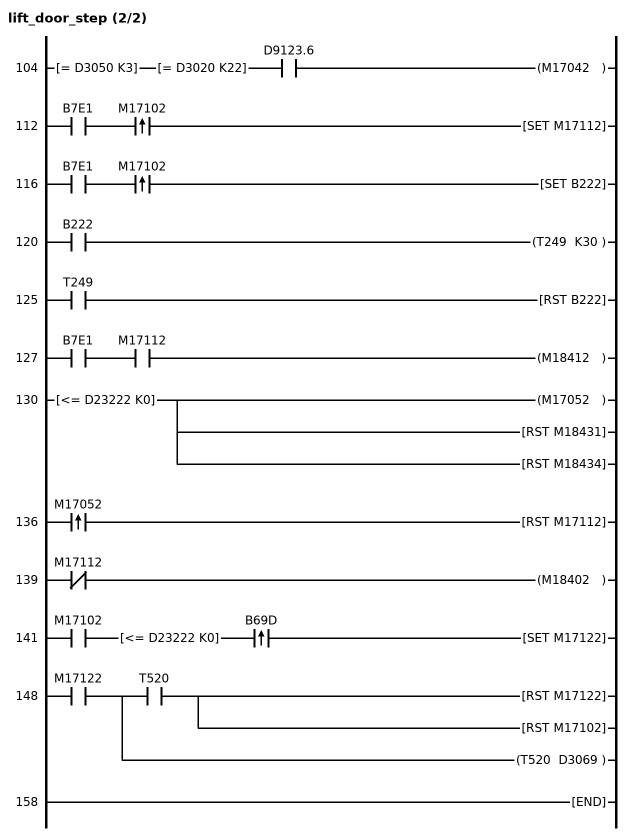
[picture p240: ladder of lift_door_step, rungs at steps 104 to 158]
104   LD=     D3050 K3
      AND=    D3020 K22
      AND     D9123.6
      OUT     M17042
112   LD      B7E1
      ANDP    M17102
      SET     M17112
116   LD      B7E1
      ANDP    M17102
      SET     B222
120   LD      B222
      OUT     T249 K30
125   LD      T249
      RST     B222
127   LD      B7E1
      AND     M17112
      OUT     M18412
130   LD<=    D23222 K0
      OUT     M17052
      RST     M18431
      RST     M18434
136   LDP     M17052
      RST     M17112
139   LDI     M17112
      OUT     M18402
141   LD      M17102
      AND<=   D23222 K0
      ANDP    B69D
      SET     M17122
148   LD      M17122
      MPS
      AND     T520
      RST     M17122
      RST     M17102
      MPP
      OUT     T520 D3069
158   END
END_PROGRAM

PROGRAM next_cap_step
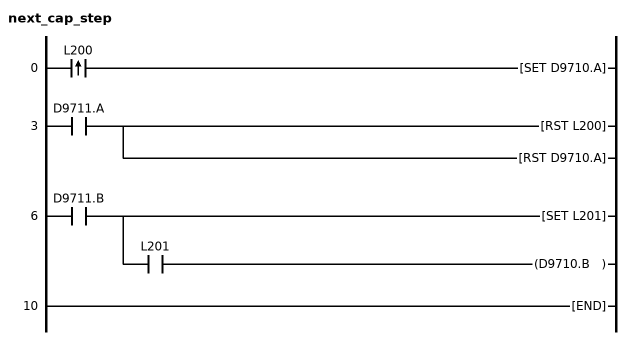
0     LDP     L200
      SET     D9710.A
3     LD      D9711.A
      RST     L200
      RST     D9710.A
6     LD      D9711.B
      SET     L201
      AND     L201
      OUT     D9710.B
10    END
END_PROGRAM

PROGRAM output
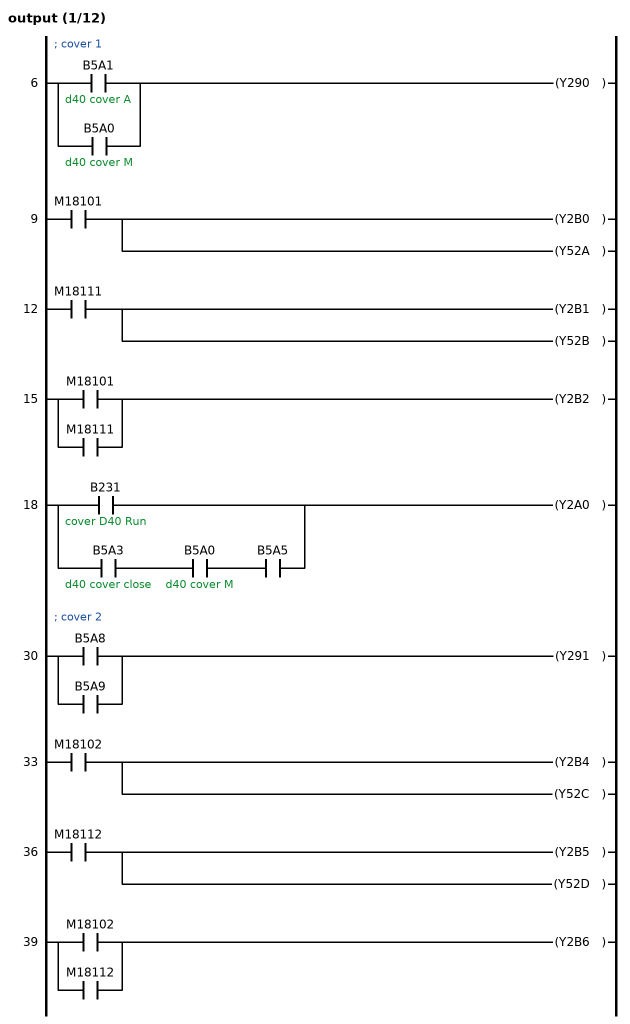
; cover 1
6     LD      B5A1  ; d40 cover A
      OR      B5A0  ; d40 cover M
      OUT     Y290
9     LD      M18101
      OUT     Y2B0
      OUT     Y52A
12    LD      M18111
      OUT     Y2B1
      OUT     Y52B
15    LD      M18101
      OR      M18111
      OUT     Y2B2
18    LD      B231  ; cover D40 Run
      LD      B5A3  ; d40 cover close
      AND     B5A0  ; d40 cover M
      AND     B5A5
      ORB
      OUT     Y2A0
; cover 2
30    LD      B5A8
      OR      B5A9
      OUT     Y291
33    LD      M18102
      OUT     Y2B4
      OUT     Y52C
36    LD      M18112
      OUT     Y2B5
      OUT     Y52D
39    LD      M18102
      OR      M18112
      OUT     Y2B6
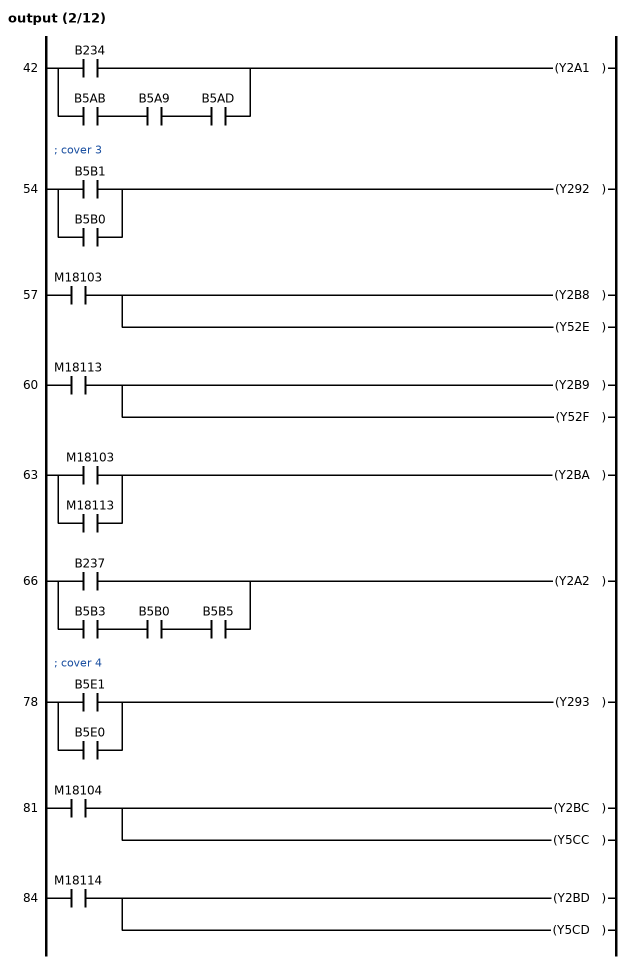
42    LD      B234
      LD      B5AB
      AND     B5A9
      AND     B5AD
      ORB
      OUT     Y2A1
; cover 3
54    LD      B5B1
      OR      B5B0
      OUT     Y292
57    LD      M18103
      OUT     Y2B8
      OUT     Y52E
60    LD      M18113
      OUT     Y2B9
      OUT     Y52F
63    LD      M18103
      OR      M18113
      OUT     Y2BA
66    LD      B237
      LD      B5B3
      AND     B5B0
      AND     B5B5
      ORB
      OUT     Y2A2
; cover 4
78    LD      B5E1
      OR      B5E0
      OUT     Y293
81    LD      M18104
      OUT     Y2BC
      OUT     Y5CC
84    LD      M18114
      OUT     Y2BD
      OUT     Y5CD
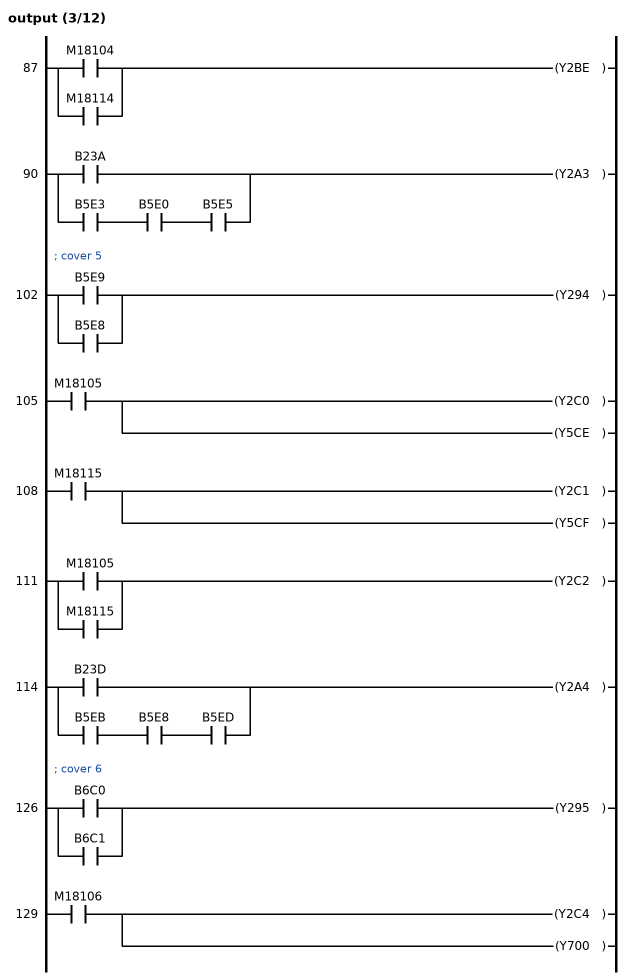
87    LD      M18104
      OR      M18114
      OUT     Y2BE
90    LD      B23A
      LD      B5E3
      AND     B5E0
      AND     B5E5
      ORB
      OUT     Y2A3
; cover 5
102   LD      B5E9
      OR      B5E8
      OUT     Y294
105   LD      M18105
      OUT     Y2C0
      OUT     Y5CE
108   LD      M18115
      OUT     Y2C1
      OUT     Y5CF
111   LD      M18105
      OR      M18115
      OUT     Y2C2
114   LD      B23D
      LD      B5EB
      AND     B5E8
      AND     B5ED
      ORB
      OUT     Y2A4
; cover 6
126   LD      B6C0
      OR      B6C1
      OUT     Y295
129   LD      M18106
      OUT     Y2C4
      OUT     Y700
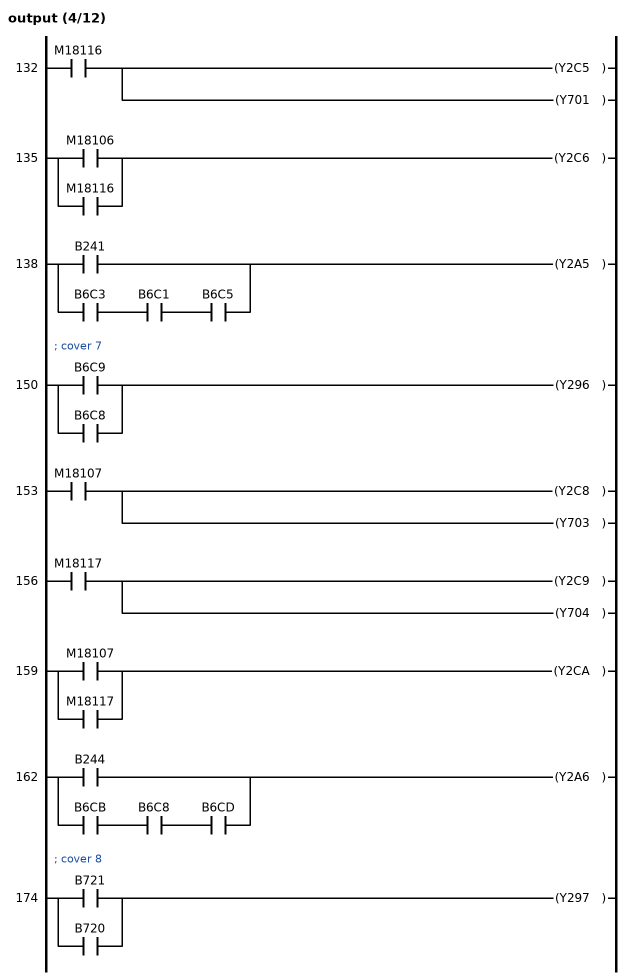
132   LD      M18116
      OUT     Y2C5
      OUT     Y701
135   LD      M18106
      OR      M18116
      OUT     Y2C6
138   LD      B241
      LD      B6C3
      AND     B6C1
      AND     B6C5
      ORB
      OUT     Y2A5
; cover 7
150   LD      B6C9
      OR      B6C8
      OUT     Y296
153   LD      M18107
      OUT     Y2C8
      OUT     Y703
156   LD      M18117
      OUT     Y2C9
      OUT     Y704
159   LD      M18107
      OR      M18117
      OUT     Y2CA
162   LD      B244
      LD      B6CB
      AND     B6C8
      AND     B6CD
      ORB
      OUT     Y2A6
; cover 8
174   LD      B721
      OR      B720
      OUT     Y297
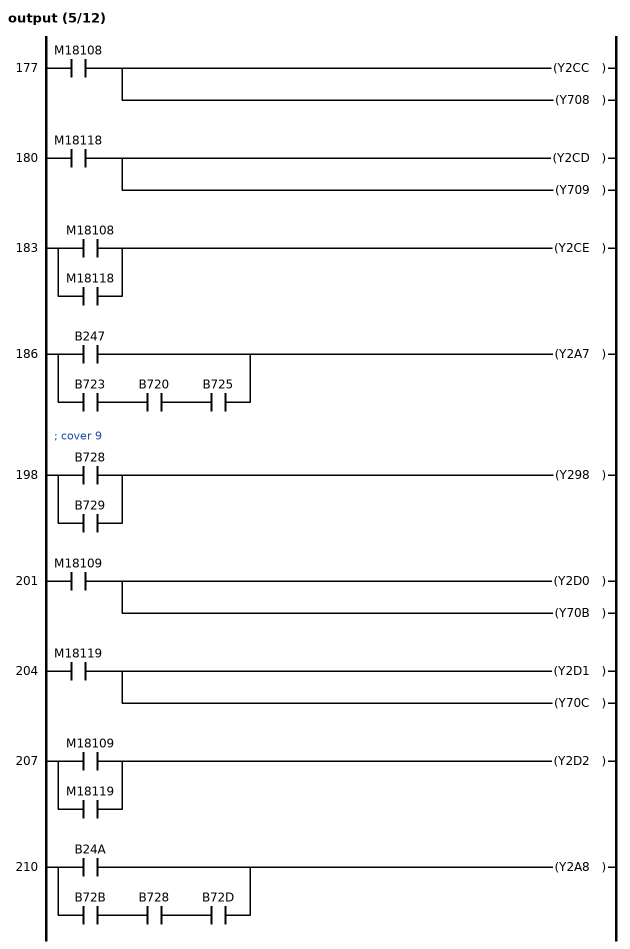
177   LD      M18108
      OUT     Y2CC
      OUT     Y708
180   LD      M18118
      OUT     Y2CD
      OUT     Y709
183   LD      M18108
      OR      M18118
      OUT     Y2CE
186   LD      B247
      LD      B723
      AND     B720
      AND     B725
      ORB
      OUT     Y2A7
; cover 9
198   LD      B728
      OR      B729
      OUT     Y298
201   LD      M18109
      OUT     Y2D0
      OUT     Y70B
204   LD      M18119
      OUT     Y2D1
      OUT     Y70C
207   LD      M18109
      OR      M18119
      OUT     Y2D2
210   LD      B24A
      LD      B72B
      AND     B728
      AND     B72D
      ORB
      OUT     Y2A8
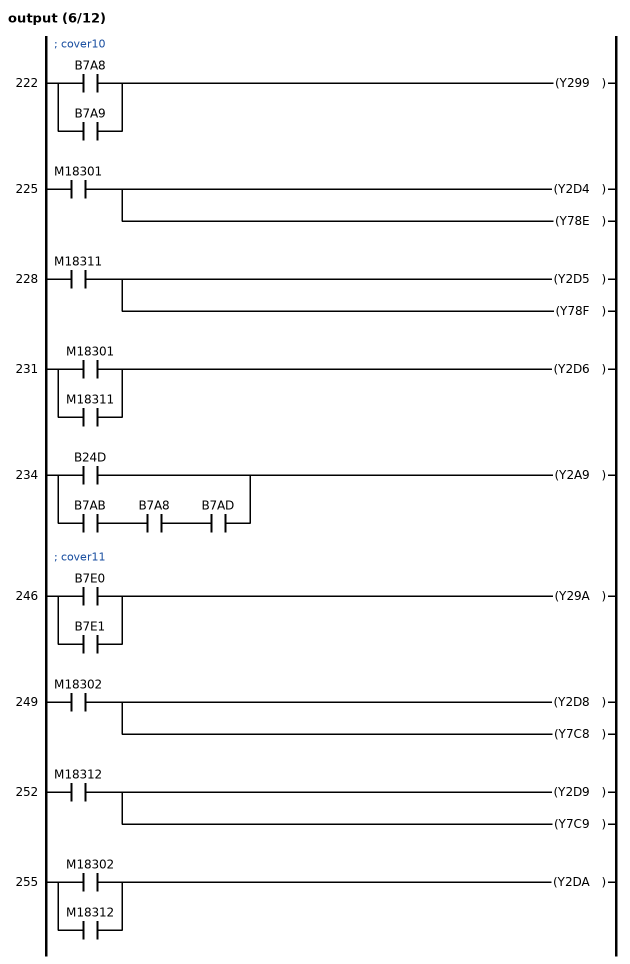
; cover10
222   LD      B7A8
      OR      B7A9
      OUT     Y299
225   LD      M18301
      OUT     Y2D4
      OUT     Y78E
228   LD      M18311
      OUT     Y2D5
      OUT     Y78F
231   LD      M18301
      OR      M18311
      OUT     Y2D6
234   LD      B24D
      LD      B7AB
      AND     B7A8
      AND     B7AD
      ORB
      OUT     Y2A9
; cover11
246   LD      B7E0
      OR      B7E1
      OUT     Y29A
249   LD      M18302
      OUT     Y2D8
      OUT     Y7C8
252   LD      M18312
      OUT     Y2D9
      OUT     Y7C9
255   LD      M18302
      OR      M18312
      OUT     Y2DA
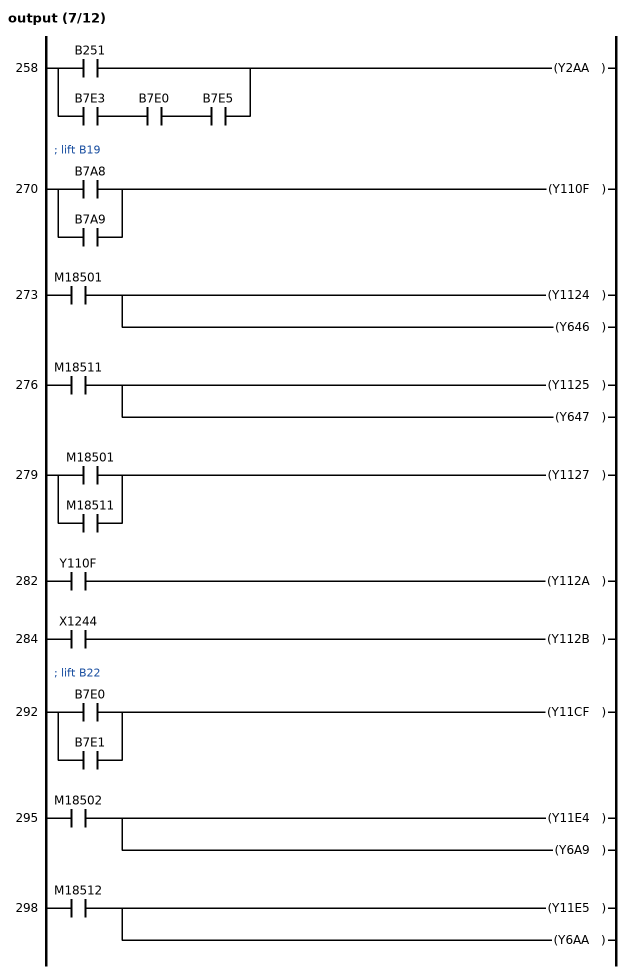
258   LD      B251
      LD      B7E3
      AND     B7E0
      AND     B7E5
      ORB
      OUT     Y2AA
; lift B19
270   LD      B7A8
      OR      B7A9
      OUT     Y110F
273   LD      M18501
      OUT     Y1124
      OUT     Y646
276   LD      M18511
      OUT     Y1125
      OUT     Y647
279   LD      M18501
      OR      M18511
      OUT     Y1127
282   LD      Y110F
      OUT     Y112A
284   LD      X1244
      OUT     Y112B
; lift B22
292   LD      B7E0
      OR      B7E1
      OUT     Y11CF
295   LD      M18502
      OUT     Y11E4
      OUT     Y6A9
298   LD      M18512
      OUT     Y11E5
      OUT     Y6AA
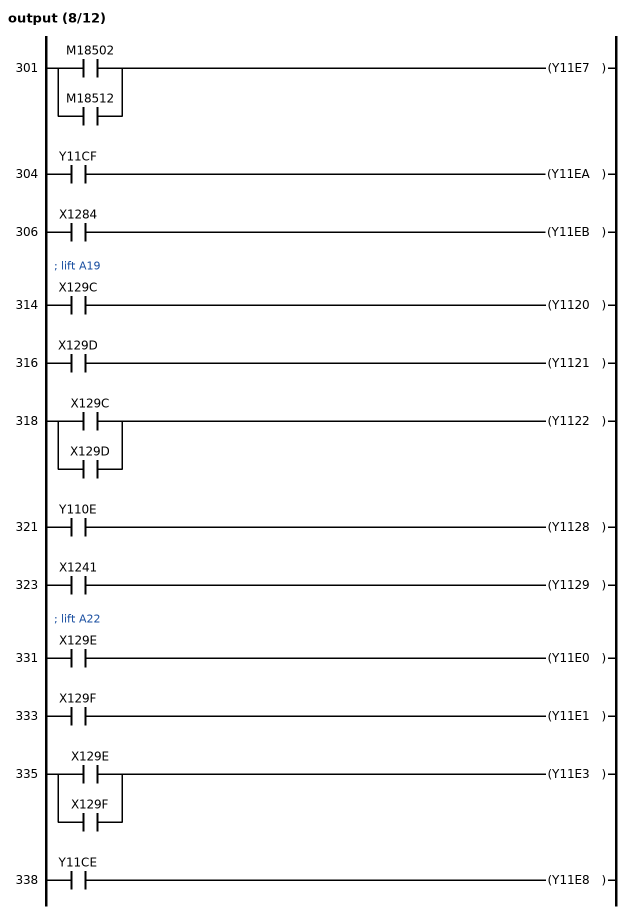
301   LD      M18502
      OR      M18512
      OUT     Y11E7
304   LD      Y11CF
      OUT     Y11EA
306   LD      X1284
      OUT     Y11EB
; lift A19
314   LD      X129C
      OUT     Y1120
316   LD      X129D
      OUT     Y1121
318   LD      X129C
      OR      X129D
      OUT     Y1122
321   LD      Y110E
      OUT     Y1128
323   LD      X1241
      OUT     Y1129
; lift A22
331   LD      X129E
      OUT     Y11E0
333   LD      X129F
      OUT     Y11E1
335   LD      X129E
      OR      X129F
      OUT     Y11E3
338   LD      Y11CE
      OUT     Y11E8
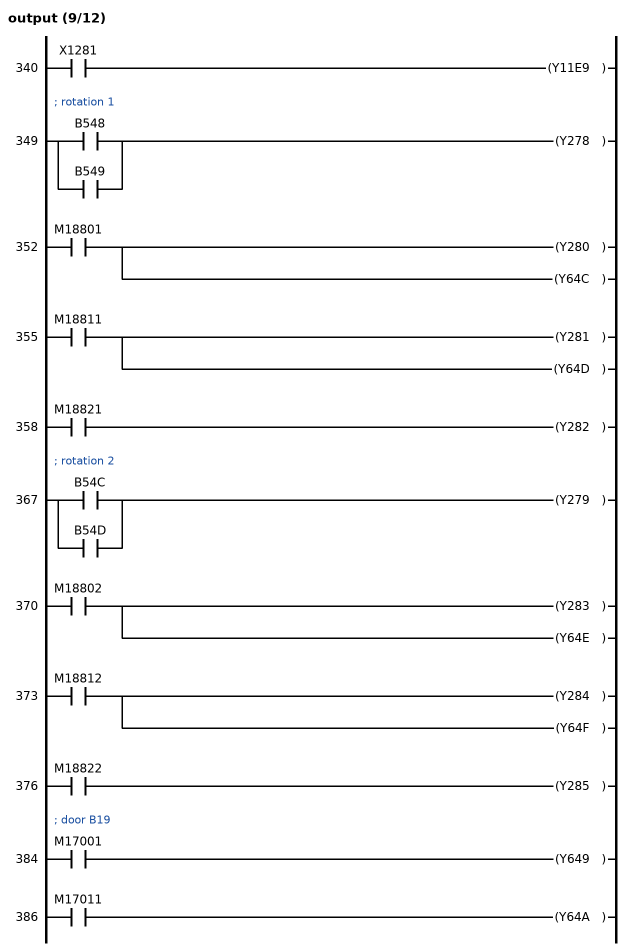
340   LD      X1281
      OUT     Y11E9
; rotation 1
349   LD      B548
      OR      B549
      OUT     Y278
352   LD      M18801
      OUT     Y280
      OUT     Y64C
355   LD      M18811
      OUT     Y281
      OUT     Y64D
358   LD      M18821
      OUT     Y282
; rotation 2
367   LD      B54C
      OR      B54D
      OUT     Y279
370   LD      M18802
      OUT     Y283
      OUT     Y64E
373   LD      M18812
      OUT     Y284
      OUT     Y64F
376   LD      M18822
      OUT     Y285
; door B19
384   LD      M17001
      OUT     Y649
386   LD      M17011
      OUT     Y64A
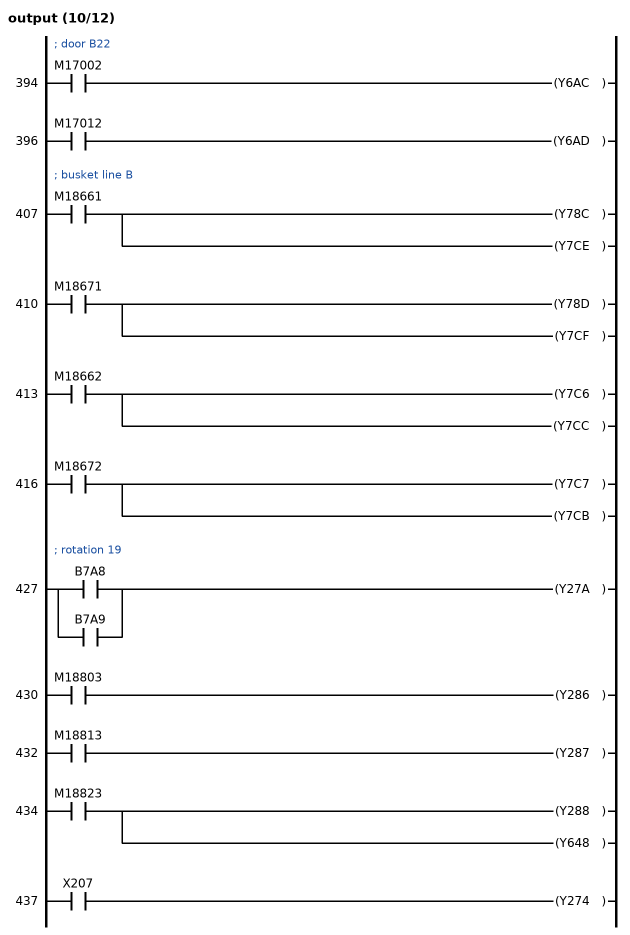
; door B22
394   LD      M17002
      OUT     Y6AC
396   LD      M17012
      OUT     Y6AD
; busket line B
407   LD      M18661
      OUT     Y78C
      OUT     Y7CE
410   LD      M18671
      OUT     Y78D
      OUT     Y7CF
413   LD      M18662
      OUT     Y7C6
      OUT     Y7CC
416   LD      M18672
      OUT     Y7C7
      OUT     Y7CB
; rotation 19
427   LD      B7A8
      OR      B7A9
      OUT     Y27A
430   LD      M18803
      OUT     Y286
432   LD      M18813
      OUT     Y287
434   LD      M18823
      OUT     Y288
      OUT     Y648
437   LD      X207
      OUT     Y274
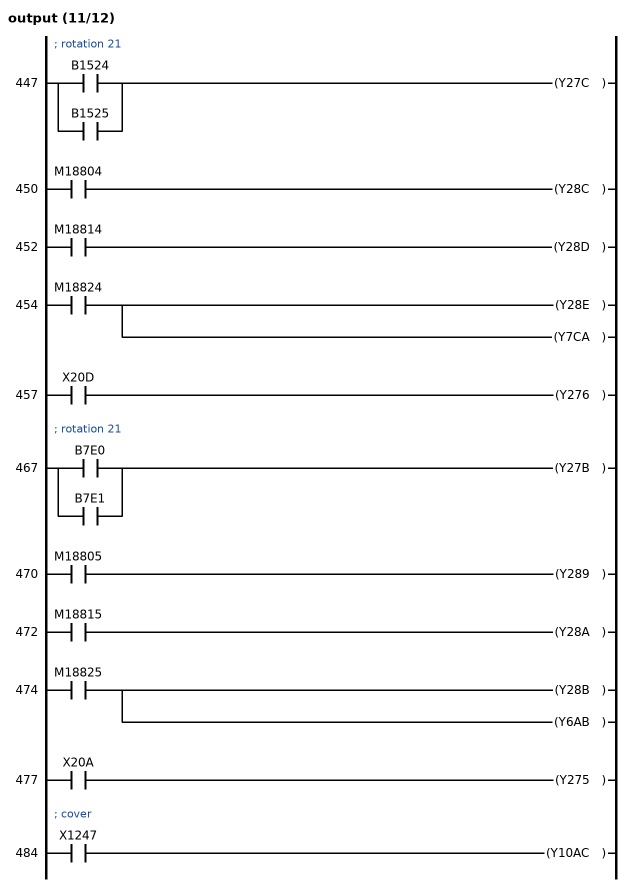
; rotation 21
447   LD      B1524
      OR      B1525
      OUT     Y27C
450   LD      M18804
      OUT     Y28C
452   LD      M18814
      OUT     Y28D
454   LD      M18824
      OUT     Y28E
      OUT     Y7CA
457   LD      X20D
      OUT     Y276
; rotation 21
467   LD      B7E0
      OR      B7E1
      OUT     Y27B
470   LD      M18805
      OUT     Y289
472   LD      M18815
      OUT     Y28A
474   LD      M18825
      OUT     Y28B
      OUT     Y6AB
477   LD      X20A
      OUT     Y275
; cover
484   LD      X1247
      OUT     Y10AC
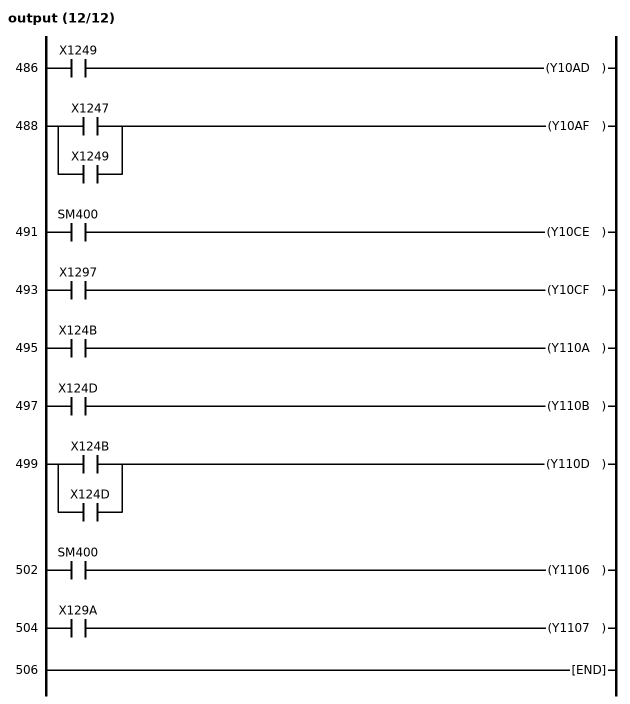
486   LD      X1249
      OUT     Y10AD
488   LD      X1247
      OR      X1249
      OUT     Y10AF
491   LD      SM400
      OUT     Y10CE
493   LD      X1297
      OUT     Y10CF
495   LD      X124B
      OUT     Y110A
497   LD      X124D
      OUT     Y110B
499   LD      X124B
      OR      X124D
      OUT     Y110D
502   LD      SM400
      OUT     Y1106
504   LD      X129A
      OUT     Y1107
506   END
END_PROGRAM

PROGRAM oven
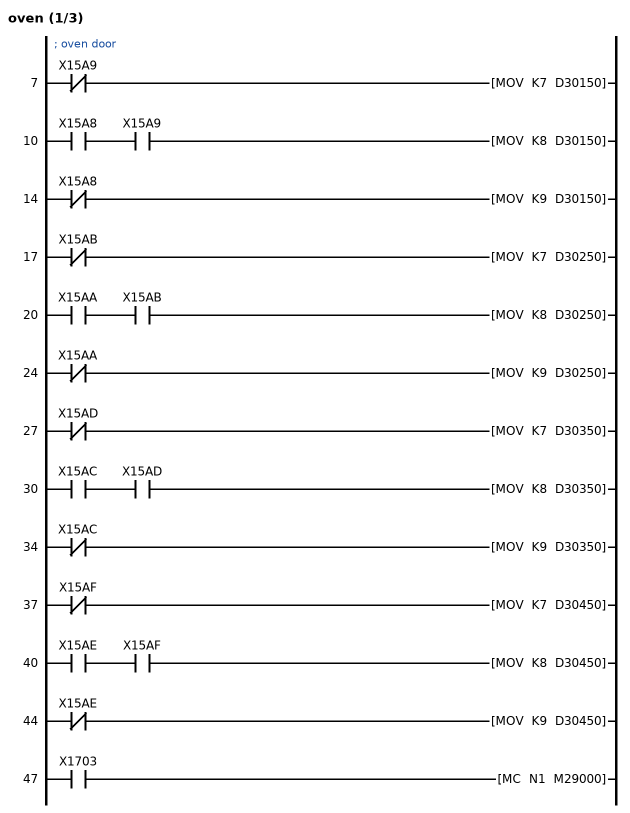
; oven door
7     LDI     X15A9
      MOV     K7 D30150
10    LD      X15A8
      AND     X15A9
      MOV     K8 D30150
14    LDI     X15A8
      MOV     K9 D30150
17    LDI     X15AB
      MOV     K7 D30250
20    LD      X15AA
      AND     X15AB
      MOV     K8 D30250
24    LDI     X15AA
      MOV     K9 D30250
27    LDI     X15AD
      MOV     K7 D30350
30    LD      X15AC
      AND     X15AD
      MOV     K8 D30350
34    LDI     X15AC
      MOV     K9 D30350
37    LDI     X15AF
      MOV     K7 D30450
40    LD      X15AE
      AND     X15AF
      MOV     K8 D30450
44    LDI     X15AE
      MOV     K9 D30450
47    LD      X1703
      MC      N1 M29000
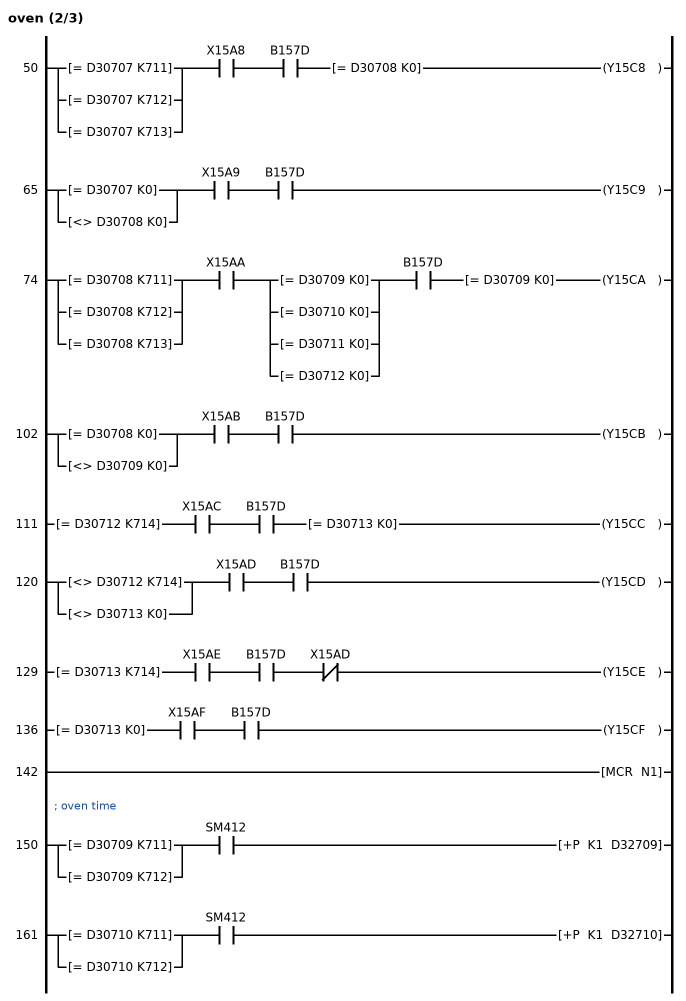
50    LD=     D30707 K711
      OR=     D30707 K712
      OR=     D30707 K713
      AND     X15A8
      AND     B157D
      AND=    D30708 K0
      OUT     Y15C8
65    LD=     D30707 K0
      OR<>    D30708 K0
      AND     X15A9
      AND     B157D
      OUT     Y15C9
74    LD=     D30708 K711
      OR=     D30708 K712
      OR=     D30708 K713
      AND     X15AA
      LD=     D30709 K0
      OR=     D30710 K0
      OR=     D30711 K0
      OR=     D30712 K0
      ANB
      AND     B157D
      AND=    D30709 K0
      OUT     Y15CA
102   LD=     D30708 K0
      OR<>    D30709 K0
      AND     X15AB
      AND     B157D
      OUT     Y15CB
111   LD=     D30712 K714
      AND     X15AC
      AND     B157D
      AND=    D30713 K0
      OUT     Y15CC
120   LD<>    D30712 K714
      OR<>    D30713 K0
      AND     X15AD
      AND     B157D
      OUT     Y15CD
129   LD=     D30713 K714
      AND     X15AE
      AND     B157D
      ANI     X15AD
      OUT     Y15CE
136   LD=     D30713 K0
      AND     X15AF
      AND     B157D
      OUT     Y15CF
142   MCR     N1
; oven time
150   LD=     D30709 K711
      OR=     D30709 K712
      AND     SM412
      +P      K1 D32709
161   LD=     D30710 K711
      OR=     D30710 K712
      AND     SM412
      +P      K1 D32710
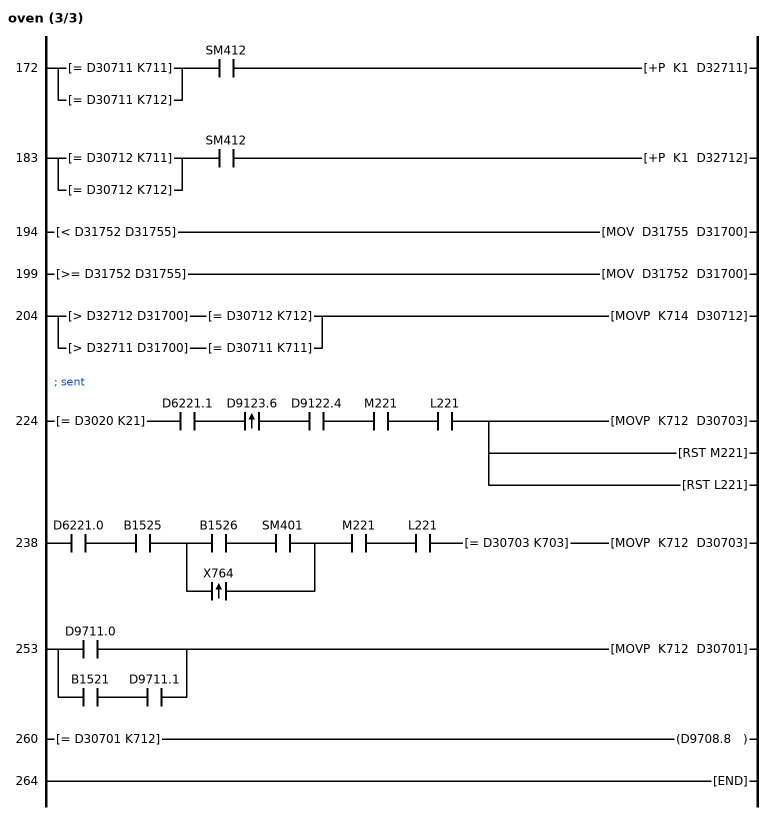
172   LD=     D30711 K711
      OR=     D30711 K712
      AND     SM412
      +P      K1 D32711
183   LD=     D30712 K711
      OR=     D30712 K712
      AND     SM412
      +P      K1 D32712
194   LD<     D31752 D31755
      MOV     D31755 D31700
199   LD>=    D31752 D31755
      MOV     D31752 D31700
204   LD>     D32712 D31700
      AND=    D30712 K712
      LD>     D32711 D31700
      AND=    D30711 K711
      ORB
      MOVP    K714 D30712
; sent
224   LD=     D3020 K21
      AND     D6221.1
      ANDP    D9123.6
      AND     D9122.4
      AND     M221
      AND     L221
      MOVP    K712 D30703
      RST     M221
      RST     L221
238   LD      D6221.0
      AND     B1525
      LD      B1526
      AND     SM401
      ORP     X764
      ANB
      AND     M221
      AND     L221
      AND=    D30703 K703
      MOVP    K712 D30703
253   LD      D9711.0
      LD      B1521
      AND     D9711.1
      ORB
      MOVP    K712 D30701
260   LD=     D30701 K712
      OUT     D9708.8
264   END
END_PROGRAM

PROGRAM POU_01
0     END
END_PROGRAM

PROGRAM pump_by_p_tongg
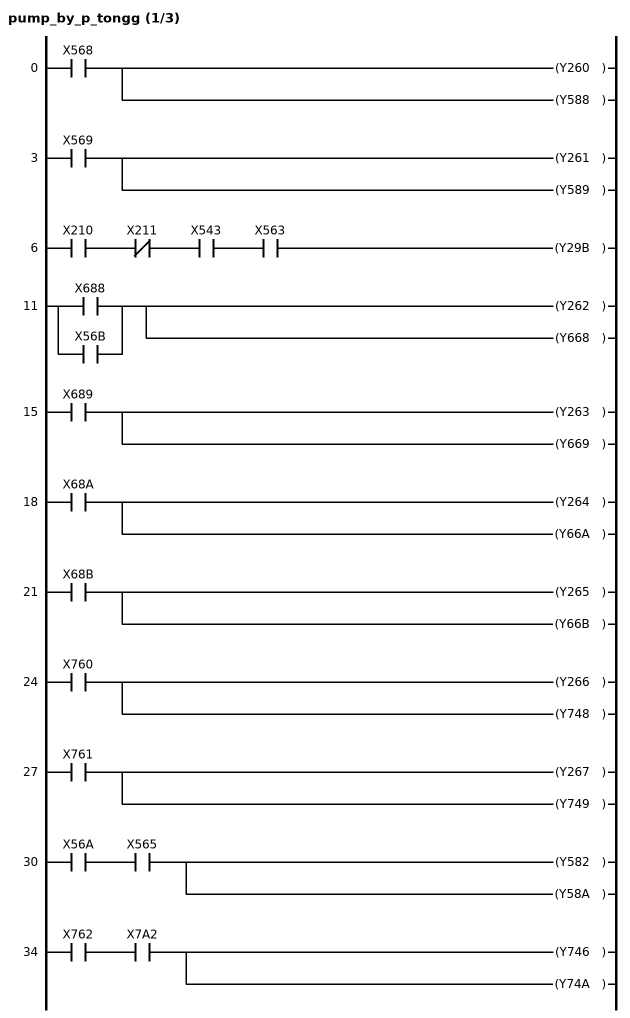
0     LD      X568
      OUT     Y260
      OUT     Y588
3     LD      X569
      OUT     Y261
      OUT     Y589
6     LD      X210
      ANI     X211
      AND     X543
      AND     X563
      OUT     Y29B
11    LD      X688
      OR      X56B
      OUT     Y262
      OUT     Y668
15    LD      X689
      OUT     Y263
      OUT     Y669
18    LD      X68A
      OUT     Y264
      OUT     Y66A
21    LD      X68B
      OUT     Y265
      OUT     Y66B
24    LD      X760
      OUT     Y266
      OUT     Y748
27    LD      X761
      OUT     Y267
      OUT     Y749
30    LD      X56A
      AND     X565
      OUT     Y582
      OUT     Y58A
34    LD      X762
      AND     X7A2
      OUT     Y746
      OUT     Y74A
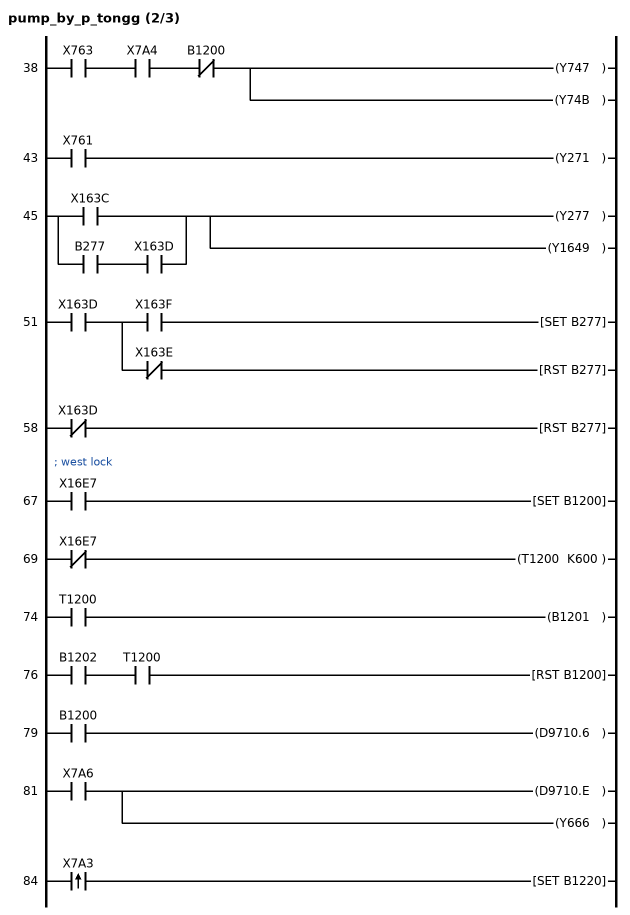
38    LD      X763
      AND     X7A4
      ANI     B1200
      OUT     Y747
      OUT     Y74B
43    LD      X761
      OUT     Y271
45    LD      X163C
      LD      B277
      AND     X163D
      ORB
      OUT     Y277
      OUT     Y1649
51    LD      X163D
      MPS
      AND     X163F
      SET     B277
      MPP
      ANI     X163E
      RST     B277
58    LDI     X163D
      RST     B277
; west lock
67    LD      X16E7
      SET     B1200
69    LDI     X16E7
      OUT     T1200 K600
74    LD      T1200
      OUT     B1201
76    LD      B1202
      AND     T1200
      RST     B1200
79    LD      B1200
      OUT     D9710.6
81    LD      X7A6
      OUT     D9710.E
      OUT     Y666
84    LDP     X7A3
      SET     B1220
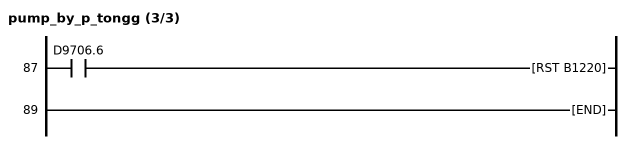
87    LD      D9706.6
      RST     B1220
89    END
END_PROGRAM

PROGRAM receive_c
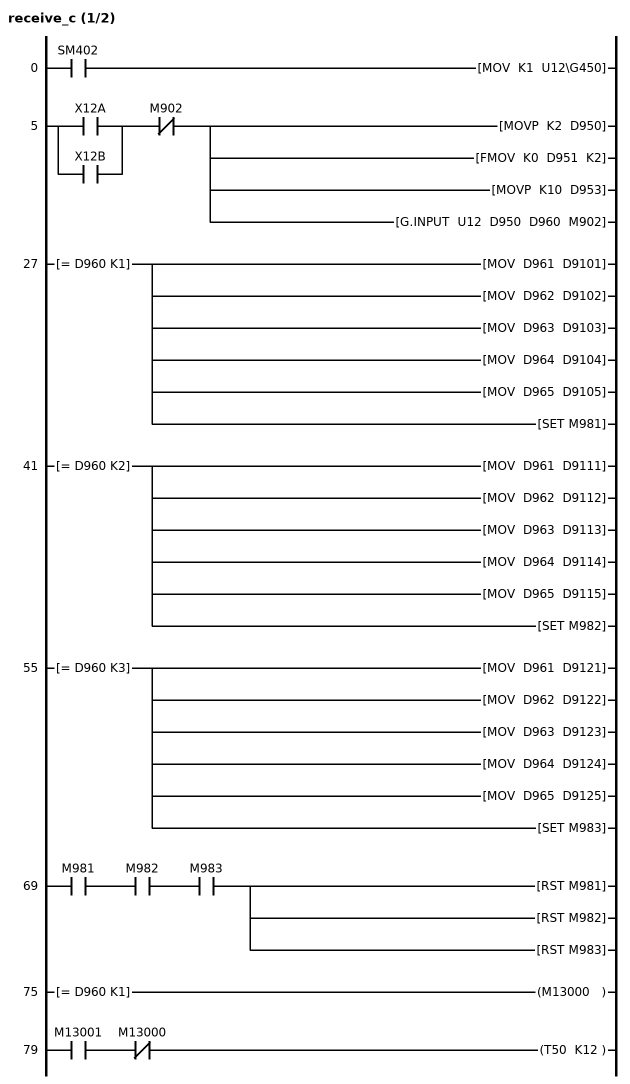
0     LD      SM402
      MOV     K1 U12\G450
5     LD      X12A
      OR      X12B
      ANI     M902
      MOVP    K2 D950
      FMOV    K0 D951 K2
      MOVP    K10 D953
      G.INPUT U12 D950 D960 M902
27    LD=     D960 K1
      MOV     D961 D9101
      MOV     D962 D9102
      MOV     D963 D9103
      MOV     D964 D9104
      MOV     D965 D9105
      SET     M981
41    LD=     D960 K2
      MOV     D961 D9111
      MOV     D962 D9112
      MOV     D963 D9113
      MOV     D964 D9114
      MOV     D965 D9115
      SET     M982
55    LD=     D960 K3
      MOV     D961 D9121
      MOV     D962 D9122
      MOV     D963 D9123
      MOV     D964 D9124
      MOV     D965 D9125
      SET     M983
69    LD      M981
      AND     M982
      AND     M983
      RST     M981
      RST     M982
      RST     M983
75    LD=     D960 K1
      OUT     M13000
79    LD      M13001
      ANI     M13000
      OUT     T50 K12
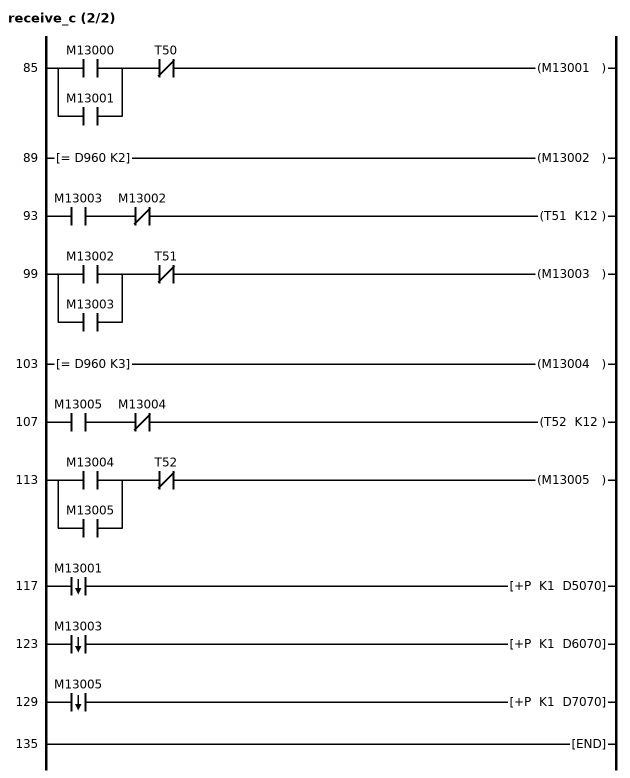
85    LD      M13000
      OR      M13001
      ANI     T50
      OUT     M13001
89    LD=     D960 K2
      OUT     M13002
93    LD      M13003
      ANI     M13002
      OUT     T51 K12
99    LD      M13002
      OR      M13003
      ANI     T51
      OUT     M13003
103   LD=     D960 K3
      OUT     M13004
107   LD      M13005
      ANI     M13004
      OUT     T52 K12
113   LD      M13004
      OR      M13005
      ANI     T52
      OUT     M13005
117   LDF     M13001
      +P      K1 D5070
123   LDF     M13003
      +P      K1 D6070
129   LDF     M13005
      +P      K1 D7070
135   END
END_PROGRAM

PROGRAM request_data
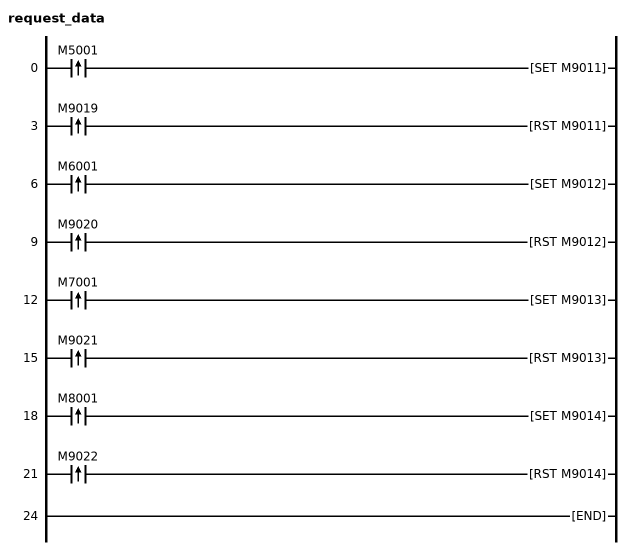
0     LDP     M5001
      SET     M9011
3     LDP     M9019
      RST     M9011
6     LDP     M6001
      SET     M9012
9     LDP     M9020
      RST     M9012
12    LDP     M7001
      SET     M9013
15    LDP     M9021
      RST     M9013
18    LDP     M8001
      SET     M9014
21    LDP     M9022
      RST     M9014
24    END
END_PROGRAM

PROGRAM rotation
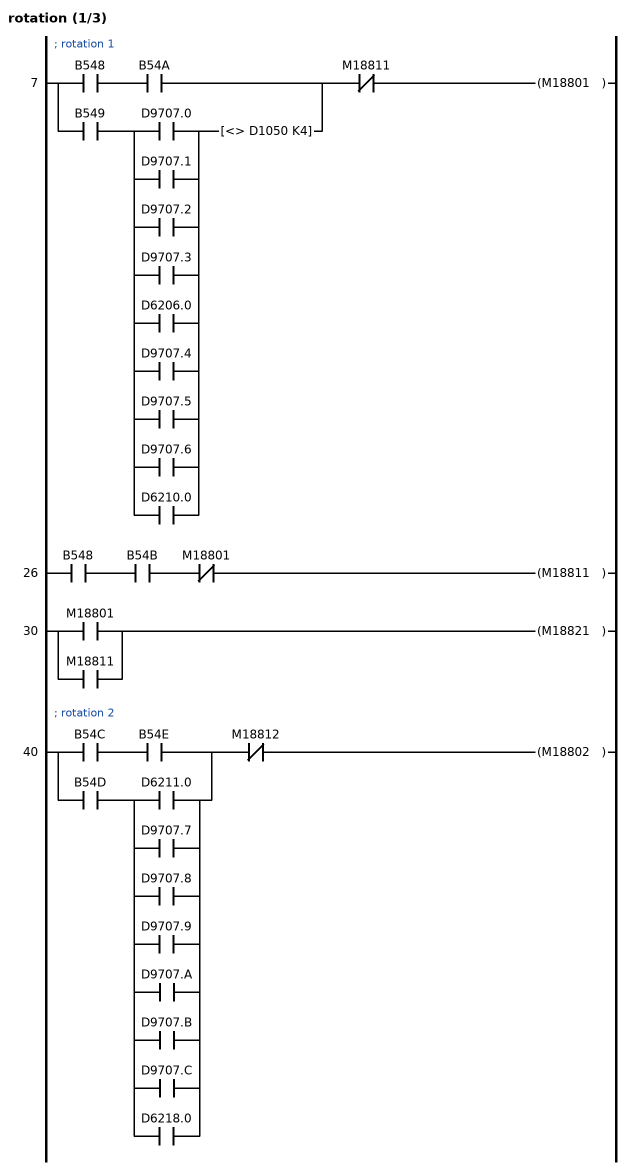
; rotation 1
7     LD      B548
      AND     B54A
      LD      B549
      LD      D9707.0
      OR      D9707.1
      OR      D9707.2
      OR      D9707.3
      OR      D6206.0
      OR      D9707.4
      OR      D9707.5
      OR      D9707.6
      OR      D6210.0
      ANB
      AND<>   D1050 K4
      ORB
      ANI     M18811
      OUT     M18801
26    LD      B548
      AND     B54B
      ANI     M18801
      OUT     M18811
30    LD      M18801
      OR      M18811
      OUT     M18821
; rotation 2
40    LD      B54C
      AND     B54E
      LD      B54D
      LD      D6211.0
      OR      D9707.7
      OR      D9707.8
      OR      D9707.9
      OR      D9707.A
      OR      D9707.B
      OR      D9707.C
      OR      D6218.0
      ANB
      ORB
      ANI     M18812
      OUT     M18802
